Fanuc KAREL source: kt00268.KL

-- PROVISIONAL review KL for V770-1; original PC SHA256 68c3c237eae649005aa70bb154173afc28fa8118c8bed81570cb4766e5eb3858
-- Incomplete behavior may be omitted. Consult companion uncertainty JSON. Do not deploy.
PROGRAM KT00268
%NOLOCKGROUP
VAR
  R2 : REAL
  OUT : BOOLEAN
-- UNRESOLVED_DECL Y1 type=002018
BEGIN
  -- UNRESOLVED_PC offsets 5-19; opcodes 2E,22,9D,33,B2
  -- UNRESOLVED_PC offsets 24-35; opcodes 2E,23
  -- UNRESOLVED_PC offsets 40-64; opcodes 22,9D,33,B1,21,29,64,6D,23
  -- UNRESOLVED_PC offsets 69-73; opcodes 7F
END KT00268
